// TwinCAT 3 PLC project Untitled1
// ProgramVersion: 3.1.4023.0
// libraries:
//   Tc2_Standard, * (Beckhoff Automation GmbH)
//   Tc2_System, * (Beckhoff Automation GmbH)
//   Tc3_Module, * (Beckhoff Automation GmbH)
// project tree:
//   GVLs/ GVL.TcGVL
//   / PlcTask.TcTTO
//   POUs/ MAIN.TcPOU
// real-time tasks:
//   TASK PlcTask: cycle T#10ms, priority 20, ADS port 350

CONFIGURATION Untitled1
    RESOURCE PLC ON TwinCAT3
        TASK PlcTask(INTERVAL := T#10ms, PRIORITY := 20);
        PROGRAM MAIN WITH PlcTask : MAIN;
    END_RESOURCE
END_CONFIGURATION

// ---- GVLs/GVL.TcGVL
{attribute 'qualified_only'}
VAR_GLOBAL
	
	{attribute 'S7.Out'}
	{attribute 'S7.Address' := 'db2.dbx0.0'}
	imAlive : BOOL;
	{attribute 'S7.In'}
	{attribute 'S7.Address' := 'db2.dbx1.0'}
	otherSystemAlive :BOOL;
	
END_VAR

// ---- POUs/MAIN.TcPOU
PROGRAM MAIN
VAR
	onTimer, offTimer : ton;
	
	start : BOOL;
END_VAR

onTimer(PT:=T#1S, Q=> GVL.imAlive);
offTimer(IN:= GVl.imAlive, PT:=T#1S);
IF offTimer.Q THEN
	onTimer.IN := FALSE;
END_IF
IF NOT GVL.imAlive AND NOT onTimer.IN THEN
	onTimer.IN := TRUE;
END_IF

END_PROGRAM
